// TIA Portal V19 export
FUNCTION "ResetAlarmBits" : Void   // FC34, STL
{ S7_Optimized_Access := 'TRUE' }
AUTHOR : FLA
FAMILY : UHT
NAME : ALAR_BIT
VERSION : 1.0
// ALAR.BIT  
// 
// Programmer Init: 8953-FLA
// 
// Change Log:
// 
// Date        Change                          Updated by
// ------------------------------------------------------
// 19.04.99    1. Edition                      FLA
// stored: AutoNumber false
BEGIN

NETWORK
TITLE = Reset alarm bits
// ;
//  Reset alarm bits
      CALL  "Alarmsystem"
      ( ONESHOT_1HZ           := "Trigger bit 1",  // 1Hz oneshot
        ALARM_DATABLOCK       := "ProcessAndPbAlarms",  // Alarm data block from functions
        ALARM_START_WORD      := 0,  // Start word 0
        NUMBER_OFF_WORDS      := 8,  // Number off words
        ALARM_COPY_DATABLOCK  := "AlarmBitScada",  // Alarm copy data block
        ALARM_COPY_START_WORD := 0,  // Start word 0
        TIME_DATA_BLOCK       := "Alarmtimer",  // Time data block
        TIME_START_WORD       := 0,  // Start word 0
        SET_ALARM_LAMP        := "Set_alarm_lamp_process"  // Set alarm lamp if new alarm
      );

NETWORK
TITLE = Reset pop up start blocking text number to intouch PC's
      CALL  "ResetPopupBlock"
      ( TRIGGER_BIT_1HZ := "Trigger bit 1"  // 1 HZ oneshot flag
      );  // Text numbers and "Count down timer" in DB36

NETWORK
TITLE = Control alarm flash lamp
      A     "OP25 TANK".Reset_lamp_Scada;  // Reset alarm flash lamp from SCADA
      R     "OP25 TANK".Reset_lamp_Scada;
      R     "Set_alarm_lamp_feedback";  // Feedback error items
      R     "Set_alarm_lamp_monitor";  // Monitor error items
      R     "Set_alarm_lamp_process";  // Process/function alarm

NETWORK
TITLE = Monitoring comm. from intouch
// If counter not change on intouch then communication alarm
      AN    "Trigger bit 1";
      JC    END4;
      L     "PopUpBitToScada".Monitor_comm_from_intouc;  // Counter comm. monitor
      L     1;  // add 1 to counter
      +I;
      T     "PopUpBitToScada".Monitor_comm_from_intouc;
END4: NOP   0;

NETWORK
TITLE = Battery low error
      A     "Alarm_battery_low_dummy";
      =     "ProcessAndPbAlarms"."A"[50];  //A50_SiemensBatteryLow// battery low


NETWORK
TITLE = FB_FAULT_VALVE_01_01
// Transfer valve alarm bits from Scada datablock to OP alarm data block
      A     "ItemInfoScada".Items["Y0101_"].fb_error;
      =     "ItemAlarmsOP".Item[1];  //FB_FAULT_VALVE_01_01
      A     "ItemInfoScada".Items[2].fb_error;
      =     "ItemAlarmsOP".Item[2];  //FB_FAULT_VALVE_01_03
      A     "ItemInfoScada".Items[3].fb_error;
      =     "ItemAlarmsOP".Item[3];  //FB_FAULT_VALVE_01_04
      A     "ItemInfoScada".Items[4].fb_error;
      =     "ItemAlarmsOP".Item[4];  //FB_FAULT_VALVE_01_09
      A     "ItemInfoScada".Items[5].fb_error;
      =     "ItemAlarmsOP".Item[5];  //FB_FAULT_VALVE_01_11
      A     "ItemInfoScada".Items[6].fb_error;
      =     "ItemAlarmsOP".Item[6];  //FB_FAULT_VALVE_01_12
      A     "ItemInfoScada".Items[7].fb_error;
      =     "ItemAlarmsOP".Item[7];  //FB_FAULT_VALVE_01_13
      A     "ItemInfoScada".Items[8].fb_error;
      =     "ItemAlarmsOP".Item[8];  //FB_FAULT_VALVE_01_14
      A     "ItemInfoScada".Items[9].fb_error;
      =     "ItemAlarmsOP".Item[9];  //FB_FAULT_VALVE_01_15
      A     "ItemInfoScada".Items[10].fb_error;
      =     "ItemAlarmsOP".Item[10];  //FB_FAULT_MOTOR_01_39
      A     "ItemInfoScada".Items[11].fb_error;
      =     "ItemAlarmsOP".Item[14];  //FB_FAULT_VALVE_01_16
      A     "ItemInfoScada".Items[12].fb_error;
      =     "ItemAlarmsOP".Item[16];  //FB_FAULT_VALVE_01_08
      A     "ItemInfoScada".Items[13].fb_error;
      =     "ItemAlarmsOP".Item[15];  //FB_FAULT_VALVE_01_17
      A     "ItemInfoScada".Items[17].fb_error;
      =     "ItemAlarmsOP".Item[17];  //FB_FAULT_VALVE_01_19
      A     "ItemInfoScada".Items[43].fb_error;
      =     "ItemAlarmsOP".Item[18];  //FB_FAULT_VALVE_WATERPUMP
//;
      A     "ItemInfoScada".Items[49].fb_error;
      =     "ItemAlarmsOP".Item[19];  //FB_FAULT_VALVE_09_04
      A     "ItemInfoScada".Items[50].fb_error;
      =     "ItemAlarmsOP".Item[20];  //FB_FAULT_VALVE_09_05
      A     "ItemInfoScada".Items[51].fb_error;
      =     "ItemAlarmsOP".Item[21];  //FB_FAULT_VALVE_09_06
      A     "ItemInfoScada".Items[52].fb_error;
      =     "ItemAlarmsOP".Item[22];  //FB_FAULT_VALVE_09_07
      A     "ItemInfoScada".Items[53].fb_error;
      =     "ItemAlarmsOP".Item[23];  //FB_FAULT_VALVE_09_08
      A     "ItemInfoScada".Items[54].fb_error;
      =     "ItemAlarmsOP".Item[24];  //FB_FAULT_VALVE_09_09
      A     "ItemInfoScada".Items[55].fb_error;
      =     "ItemAlarmsOP".Item[25];  //FB_FAULT_VALVE_09_10
      A     "ItemInfoScada".Items[56].fb_error;
      =     "ItemAlarmsOP".Item[26];  //FB_FAULT_VALVE_09_11
      A     "ItemInfoScada".Items[57].fb_error;
      =     "ItemAlarmsOP".Item[27];  //FB_FAULT_VALVE_09_12
//;
      A     "IF_Device".V_09_30.IO.V._IO.IN_OUT.HMI_INFO.%X14;
      =     "ItemAlarmsOP".Item[28];  //FB_FAULT_VALVE_09_30
      A     "IF_Device".V_09_31.IO.V._IO.IN_OUT.HMI_INFO.%X14;
      =     "ItemAlarmsOP".Item[29];  //FB_FAULT_VALVE_09_31

END_FUNCTION
